{attribute 'qualified_only'}
VAR_GLOBAL
// Glovel Bit
	Pulse_100ms					:	BOOL	;			//0.1s Bit
	Pulse_1S					:	BOOL	;			//1S Bit		
// System Bit
	Manual_Mode					:	BOOL	;			//HMI 메뉴얼 모드
	Auto_Mode					:	BOOL	;			//HMI 오토모드
	Stop						:	BOOL	;			//HMI Stop
	Safety_ALL_OK				:	BOOL	;			//EMO+Door
	Test_Mode					:	BOOL	;
	All_Initial					:	BOOL	;
//EMO SW	
	EMO_SWitch		AT%I*		:	BOOL	;
//Fiber Sensor
	Vision_Start_Sensor	AT%I*	:	BOOL	;
	Press_Start_Sensor	AT%I*	:	BOOL	;
	Press_End_Sensor	AT%I*	:	BOOL	;

//System_Door_Sensor
	Door_Open					:	BOOL	;

//TowerLamp
	Tower_Lamp_Green	AT%Q*	:	BOOL	;
	Tower_Lamp_Yellow	AT%Q*	:	BOOL	;
	Tower_Lamp_Red		AT%Q*	:	BOOL	;
	Buzzer				AT%Q*	:	BOOL	;
//HMI
	Buzzer_Stop					:	BOOL	;
	Alarm_Reset					:	BOOL	;
//Panel
	DC01_SMPS_OK					AT%I*	:	BOOL	;
	DC02_SMPS_OK					AT%I*	:	BOOL	;
	DC03_SMPS_OK					AT%I*	:	BOOL	;
	Servo_Drive_Control_DC_Power	AT%I*	:	BOOL	;
	HUB_Power_OK					AT%I*	:	BOOL	;
	
//Bool
	HMI_Auto_Mode				:	BOOL	;		//HMI 오토모드
	ALL_Motor_Homed				:	BOOL	;		//전체 모터 홈 OK
	ALL_Motor_Home_Position		:	BOOL	;		//전체 모터 홈포지션
	HMI_Manual_Mode				:	BOOL	;		//HMI 메뉴얼 모드
	ALL_Motor_Busy				:	BOOL	;		//전체 모터 동작중
	ALL_Motor_StandStill		:	BOOL	;		//전체 모터 동작 가능
	Moving_Motor_Wait_Position	:	BOOL	;		//X,Y,Z,R Wait Position
	Each_Motor_Homed			:	BOOL	;		//개별 로못 홈
	Each_Motor_Busy				:	BOOL	;		//개별 로봇 동작중
	All_Motor_Stop				:	BOOL	;	
	
	
	
	Test_Data_Read_Comp			: 	BOOL	;
	Test_Continues				: 	BOOL	;
	Calibration_Mode			: 	BOOL	;
	Tool_Change_Mode			: 	BOOL	;
	Tool_Change_Move_PB			: 	BOOL	;	
//홈동작 
	ALL_Wait_Position			: 	BOOL	;
	ALL_Home_Move_PB			:	BOOL	;
	ALL_Home_Move_Start			:	BOOL	;
	Axis01_Home_Move			: 	BOOL	;
	Axis02_Home_Move			: 	BOOL	;
	Axis03_Home_Move			: 	BOOL	;
	Axis04_Home_Move			: 	BOOL	;
	Axis05_Home_Move			: 	BOOL	;
	
	Axis01_Home_Pos_Move		: 	BOOL	;
	Axis04_Wait_Pos_Move		:	BOOL	;
	Axis03_Wait_Pos_Move		: 	BOOL	;
	Axis01_Wait_Pos_Move		: 	BOOL	;
	Axis02_Wait_Pos_Move		: 	BOOL	;
	Axis05_Wait_Pos_Move		: 	BOOL	;	
	Calibration_PB: BOOL;
	Test_Start: BOOL;
END_VAR

(* stored: Version 1.1.0.1, ProductVersion 3.1.4024.15
   GVL GVL_System_1: Id {0c323435-7485-449c-8bfc-1d18c5952621} *)
